PROGRAM MAIN
VAR
	var1	: UINT;
	var2	: LREAL;
	var3	: STRING;
	var4	: BOOL;
	var5	: ARRAY[0..999] OF T_MaxString;
	var6	: ARRAY[0..2] OF dt_params;

END_VAR


//just commands to the slow task
recipes.load;
recipes.save;
recipes.count;
recipes.delete;
recipes.name;
recipes.result;

END_PROGRAM

(* stored: Version 1.1.0.1, ProductVersion 3.1.4026.12
   POU MAIN: Id {b5584c18-0e6b-42fb-8ba8-96aa3f08675c}, SpecialFunc None *)
